// TIA Portal V20 export
DATA_BLOCK "ALARM"   // DB800
{ S7_Optimized_Access := 'FALSE' }
VERSION : 0.1
// stored: AutoNumber false, DBAccessibleFromOPCUA true, DBAccessibleFromWebserver true, IsOnlyStoredInLoadMemory false, IsWriteProtectedInAS false
   VAR
      FAULT : Array[0..399] of Byte;
      WARN : Array[0..399] of Byte;
      EVENT : Array[0..31] of Byte;   // Operator (ErrorList O), byte / bit = number rule
      INFO : Array[0..39] of Byte;   // Info (ErrorList I)
   END_VAR
BEGIN
END_DATA_BLOCK
